FUNCTION_BLOCK FB_Coordinador_SFC

VAR_IN_OUT
	CiclosPendientes: UINT;
	CiclosAceptados: UINT;
END_VAR
VAR_INPUT
	// SFC-Flags
    SFCPause: BOOL;
    SFCReset: BOOL;
    
    // Indicadores de sincronizacion
    Ack: BOOL := TRUE;
    Execute: BOOL;
    
    // Parametros de sincronizacion
    PaleSituado: BOOL;
    Verificado: BOOL;
	Rechazado: BOOL;
    BaseCargada: BOOL;
    PaleTransferido: BOOL;
    
    // Parametros
    CondicionInicial: BOOL;
    CiclosSolicitados: UINT;
END_VAR
VAR_OUTPUT
	// Indicadores de sincronizacion
    Done: BOOL;
    Ready: BOOL;

    // Parametros de sincronizacion
    SituaPale: BOOL;
    VerificaBase: BOOL;
    RechazaBase: BOOL;
	CargaBase: BOOL;
    TransfierePale: BOOL;
    
    // Salidas
    LamparaAlarma: BOOL;
    LamparaMarcha: BOOL;
END_VAR
VAR
	// Bloques funcionales
    CLK: FB_Clock;
	//Entradas
	Base_en_Alimentador AT %I*: BOOL;
END_VAR

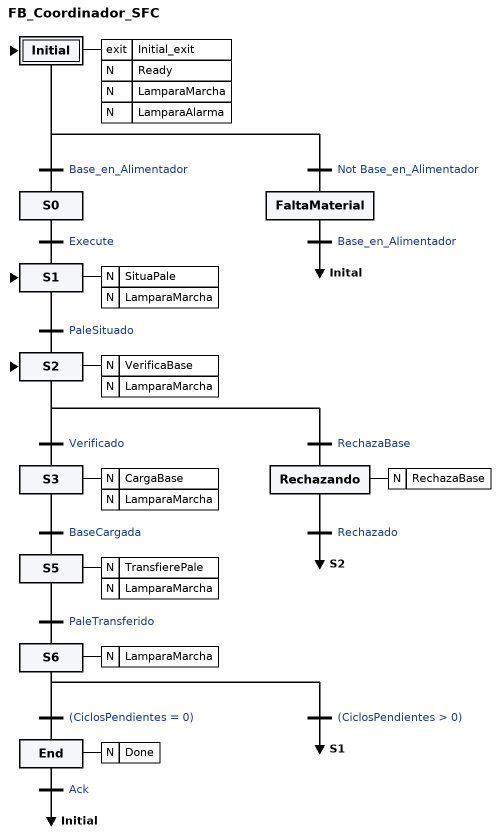
INITIAL_STEP Initial:
    Initial_exit(P0);  // exit action
    Ready(N);
    LamparaMarcha(N);
    LamparaAlarma(N);
END_STEP
TRANSITION FROM Initial TO S0
    := Base_en_Alimentador;
END_TRANSITION
STEP S0:
END_STEP
TRANSITION FROM Initial TO FaltaMaterial
    := Not Base_en_Alimentador;
END_TRANSITION
STEP FaltaMaterial:
END_STEP
TRANSITION FROM FaltaMaterial TO Inital
    := Base_en_Alimentador;
END_TRANSITION
TRANSITION FROM S0 TO S1
    := Execute;
END_TRANSITION
STEP S1:
    SituaPale(N);
    LamparaMarcha(N);
END_STEP
TRANSITION FROM S1 TO S2
    := PaleSituado;
END_TRANSITION
STEP S2:
    VerificaBase(N);
    LamparaMarcha(N);
END_STEP
TRANSITION FROM S2 TO S3
    := Verificado;
END_TRANSITION
TRANSITION FROM S2 TO Rechazando
    := RechazaBase;
END_TRANSITION
STEP Rechazando:
    RechazaBase(N);
END_STEP
TRANSITION FROM Rechazando TO S2
    := Rechazado;
END_TRANSITION
STEP S3:
    CargaBase(N);
    LamparaMarcha(N);
END_STEP
TRANSITION FROM S3 TO S5
    := BaseCargada;
END_TRANSITION
STEP S5:
    TransfierePale(N);
    LamparaMarcha(N);
END_STEP
TRANSITION FROM S5 TO S6
    := PaleTransferido;
END_TRANSITION
STEP S6:
    LamparaMarcha(N);
END_STEP
TRANSITION FROM S6 TO End
    := (CiclosPendientes = 0);
END_TRANSITION
TRANSITION FROM S6 TO S1
    := (CiclosPendientes > 0);
END_TRANSITION
STEP End:
    Done(N);
END_STEP
TRANSITION FROM End TO Initial
    := Ack;
END_TRANSITION

ACTION Initial_exit:
IF (CiclosPendientes = 0) THEN
	CiclosPendientes := CiclosSolicitados;
END_IF
END_ACTION

END_FUNCTION_BLOCK

(* stored: Version 1.1.0.1, ProductVersion 3.1.4024.12
   POU FB_Coordinador_SFC: Id {71b93a32-98c3-40e8-882e-9ce7bdbace69}, SpecialFunc None
   Action Initial_exit: Id {8ec35d20-aecc-4d29-aefd-5a57190ef6fe} *)
